Staubli VAL3: STRALIGN.pgx

public program strAlign(string& x_sStrIn[], num x_nLength, string x_sAlign, string x_sChar)
  local num l_i
  local num l_nToAdd
  local num l_nAscii
begin
  // This program modify the input string to align it
  // left,right or centered
  //
  // Input Param
  // x_sStrIn   : Input string to modify
  // x_nLength  : Length of the output string
  // x_sAlign   : Align mode
  //                  : C-c = Centered
  //                    L-l = Align Left
  //                    R-r = Align Right
  //Created 13/03/04                              C.CURRIVAND
  //--------------------------------------------------------------
  switch asc(x_sAlign,0)
    // Centered
    case 67,99
    break
    // Left
    case 76,108
      if len(x_sStrIn)<x_nLength
        l_nToAdd=x_nLength-len(x_sStrIn)
        for l_i=1 to l_nToAdd
          x_sStrIn=x_sStrIn+x_sChar
        endFor
      else
        x_sStrIn=mid(x_sStrIn,x_nLength,0)
      endIf
    break
    // Right
    case 82,114
      if len(x_sStrIn)<x_nLength
        l_nToAdd=x_nLength-len(x_sStrIn)
        for l_i=1 to l_nToAdd
          x_sStrIn=x_sChar+x_sStrIn
        endFor
      else
        x_sStrIn=mid(x_sStrIn,x_nLength,0)
      endIf
    break
  endSwitch
end
